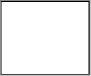
VISUALIZATION VISU_HMI_SYSTEM_BUTTON  // 91x76
VAR_IN_OUT
    m_Hmi : FB_HMI_BUTTON;
END_VAR
    Rectangle (0,0 90x75), invisible if: m_Hmi.bIsNotOrange
    Rectangle (0,0 90x75), invisible if: m_Hmi.bIsNotGray
    Rectangle (0,0 90x75), invisible if: m_Hmi.bIsNotBlue
    Rectangle (0,0 90x75), invisible if: m_Hmi.bIsNotRed
    Rectangle (0,0 90x75), invisible if: m_Hmi.bIsNotGreen
    Rectangle (0,50 90x25), "%s", text variable: m_Hmi.sName
    Image (25,10 40x40), image: VISU_HMI_BUTTON_IMAGES.Start
        p84334746: m_Hmi.sIconName
    Rectangle (0,0 90x75), invisible if: m_Hmi.bNotActivated
    Line (0,74) (90,74), invisible if: m_Hmi.bActivated
    Line (89,75) (89,0), invisible if: m_Hmi.bActivated
    Line (0,74) (0,0), invisible if: m_Hmi.bActivated
    Line (88,0) (0,0), invisible if: m_Hmi.bActivated
    Line (0,1) (90,1), invisible if: m_Hmi.bNotActivated
    Line (1,75) (1,0), invisible if: m_Hmi.bNotActivated
    Line (90,75) (1,75), invisible if: m_Hmi.bNotActivated
    Line (90,75) (90,1), invisible if: m_Hmi.bNotActivated
END_VISUALIZATION

(* stored: Version 1.1.0.1, ProductVersion 3.1.4024.14
   Visu VISU_HMI_SYSTEM_BUTTON: Id {66dc4bb4-f1df-4ee3-93ae-3509e249ae72} *)
